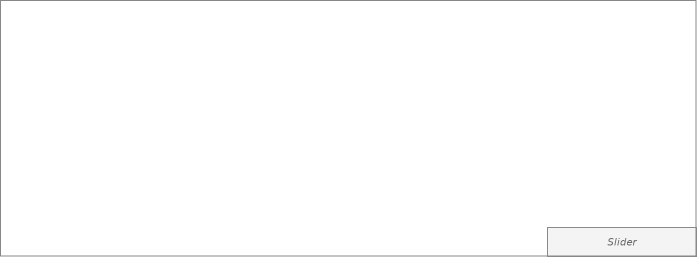
VISUALIZATION Visualization  // 697x257
    Slider (547,227 150x30), variable: MAIN.linearVel, scale 0..20000
END_VISUALIZATION

(* stored: Version 1.1.0.1, ProductVersion 3.1.4024.12
   Visu Visualization: Id {b4cb83ea-630f-4277-bd85-3a3c82211252} *)
